PROGRAM MAIN
VAR
END_VAR

END_PROGRAM

(* stored: Version 1.1.0.1
   POU MAIN: Id {3526f935-dced-4bd8-a362-3d0b59da9f6c} *)
